TYPE "UDT_HMI_Alarm_V2"
VERSION : 0.1
   STRUCT
      t : Struct
         x0 : Bool;
         x1 : Bool;
         x2 : Bool;
         x3 : Bool;
         x4 : Bool;
         x5 : Bool;
         x6 : Bool;
         x7 : Bool;
         x8 : Bool;
         x9 : Bool;
         x10 : Bool;
         x11 : Bool;
         x12 : Bool;
         x13 : Bool;
         x14 : Bool;
         x15 : Bool;
      END_STRUCT;
      iHmiSumAlm : Word;
   END_STRUCT;

END_TYPE

TYPE "UDT_Conveyor_Hmi_V0.01"
VERSION : 0.1
   STRUCT
      tHMR { ExternalWritable := 'False'} : Struct   // {[Unit]|[Scada Unit]|[LowLimit]|[HigLimit]|[Acces]}
         xManualCommandEnabled { ExternalWritable := 'False'} : Bool;   // Manual Mode Enable {x|x|x|x|O}
         xVirtualDoorEnabled { ExternalWritable := 'False'} : Bool;   // Virtual Door Enable {x|x|x|x|O}
         xCleaningEnabled { ExternalWritable := 'False'} : Bool;   // Cleaning Enabled {x|x|x|x|O}
         xPlatePresence { ExternalWritable := 'False'} : Bool;   // Plate Present {x|x|x|x|O}
         iState { ExternalWritable := 'False'} : Int;   // State (1=No anomaly, 3=Run, 7=Anomaly) {x|x|x|x|O}
         iStateMotor { ExternalWritable := 'False'} : Array["STARTARRAY".."DNMOTORCONV"] of Int;
         tManCmd { ExternalWritable := 'False'} : Struct
            xCmdFwd { ExternalWritable := 'False'} : Bool;   // Manual Command Fwd{x|x|x|x|O}
            xCmdBkw { ExternalWritable := 'False'} : Bool;   // Manual Command Bkw {x|x|x|x|O}
         END_STRUCT;
      END_STRUCT;
      tHMW : Struct   // {[Unit]|[Scada Unit]|[LowLimit]|[HigLimit]|[Acces]}
         xLocalCleaningRequest : Bool;   // Cleaning Request {x|x|x|x|O}
         xEnableDisableManualCommand : Bool;   // Enable/Disable manual command{x|x|x|x|O}
         xEnableVirtualDoor : Bool;   // Enable/Disable virtual door{x|x|x|x|O}
         tManCmd : Struct
            xCmdFwd : Bool;   // Manual Command Rise {x|x|x|x|O}
            xCmdBkw : Bool;   // Manual Command Descend{x|x|x|x|O}
         END_STRUCT;
      END_STRUCT;
   END_STRUCT;

END_TYPE

DATA_BLOCK "Conveyor_Alm"
{ S7_Optimized_Access := 'FALSE' }
VERSION : 0.1
   STRUCT
      rgtInd : Array["STARTARRAY".."DNMCONVEYOR"] of Struct
         tEmergencyAlarm { ExternalWritable := 'False'} : Array["STARTARRAY".."DALARM"] of "UDT_HMI_Alarm_V2";
         tAlarm { ExternalWritable := 'False'} : Array["STARTARRAY".."DALARM"] of "UDT_HMI_Alarm_V2";
         tWarning { ExternalWritable := 'False'} : Array["STARTARRAY".."DALARM"] of "UDT_HMI_Alarm_V2";
      END_STRUCT;
   END_STRUCT;


BEGIN

END_DATA_BLOCK

DATA_BLOCK "Conveyor_hmi"
{ S7_Optimized_Access := 'FALSE' }
VERSION : 0.1
   STRUCT
      rgtInd : Array["STARTARRAY".."DNMCONVEYOR"] of "UDT_Conveyor_Hmi_V0.01";
   END_STRUCT;


BEGIN

END_DATA_BLOCK

